FUNCTION_BLOCK DistStnArm (* Basic Function Block Type *)
  (* Standard: 61499-2 *)
  (* Version 0.2, 2003-12-04, JHC, Rockwell Automation, Renamed for better indexing. *)
  (* Compiler header: package fb.rt.wago; #include <sys/time.h> *)
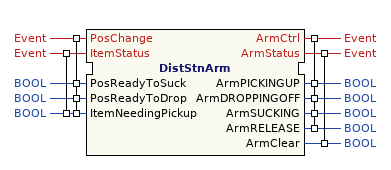
  EVENT_INPUT
    PosChange WITH PosReadyToSuck, PosReadyToDrop, ItemNeedingPickup; (* Normal Execution Request *)
    ItemStatus WITH ItemNeedingPickup;
  END_EVENT
  EVENT_OUTPUT
    ArmCtrl WITH ArmPICKINGUP, ArmDROPPINGOFF, ArmSUCKING, ArmRELEASE;
    ArmStatus WITH ArmClear; (* Execution Confirmation *)
  END_EVENT
  VAR_INPUT
    PosReadyToSuck : BOOL := false; (* Input event qualifier *)
    PosReadyToDrop : BOOL := false; (* Input event qualifier *)
    ItemNeedingPickup : BOOL;
  END_VAR
  VAR_OUTPUT
    ArmPICKINGUP : BOOL := false;
    ArmDROPPINGOFF : BOOL := false; (* Output event qualifier *)
    ArmSUCKING : BOOL := false;
    ArmRELEASE : BOOL := false;
    ArmClear : BOOL := true;
  END_VAR
  VAR
    ReleaseDelay : INT;
  END_VAR
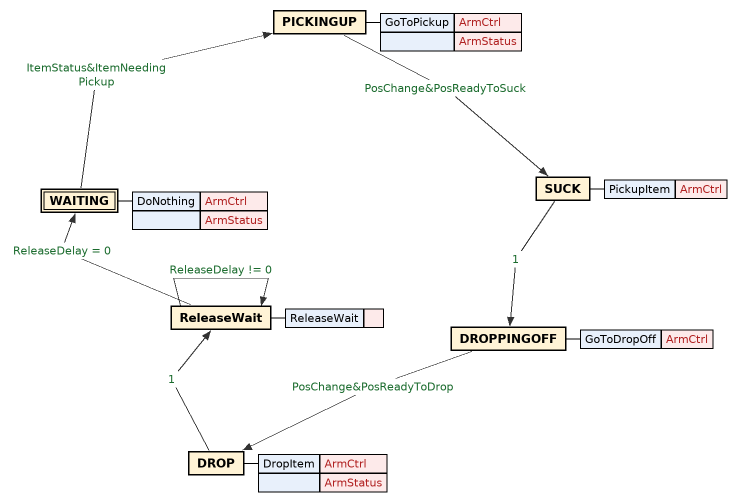
  EC_STATES
    WAITING : DoNothing -> ArmCtrl, -> ArmStatus; (* Initial State *)
    DROPPINGOFF : GoToDropOff -> ArmCtrl; (* Normal execution *)
    DROP : DropItem -> ArmCtrl, -> ArmStatus; (* Normal execution *)
    PICKINGUP : GoToPickup -> ArmCtrl, -> ArmStatus;
    SUCK : PickupItem -> ArmCtrl;
    ReleaseWait : ReleaseWait;
  END_STATES
  EC_TRANSITIONS
    WAITING TO PICKINGUP := ItemStatus&ItemNeedingPickup;
    PICKINGUP TO SUCK := PosChange&PosReadyToSuck;
    SUCK TO DROPPINGOFF := 1;
    DROPPINGOFF TO DROP := PosChange&PosReadyToDrop;
    DROP TO ReleaseWait := 1;
    ReleaseWait TO WAITING := ReleaseDelay = 0;
    ReleaseWait TO ReleaseWait := ReleaseDelay != 0;
  END_TRANSITIONS
  ALGORITHM GoToDropOff IN C: (* Initialization algorithm *)
me->ArmPICKINGUP = false;
me->ArmDROPPINGOFF = true;
  END_ALGORITHM
  ALGORITHM GoToPickup IN C: (* Initialization algorithm *)
me->ArmPICKINGUP = true;
me->ArmDROPPINGOFF = false;

me->ArmClear = false;
  END_ALGORITHM
  ALGORITHM PickupItem IN C: (* Normally executed algorithm *)
me->ArmSUCKING = true;
me->ArmRELEASE = false;
  END_ALGORITHM
  ALGORITHM CheckTimeout IN C:
//struct timeval nowtime, timediff;
//long long result;

//gettimeofday(&nowtime, NULL);
//timersub(&nowtime, &me->armTimer, &timediff);
//result = (long long)(timediff.tv_sec) * 1000000 + timediff.tv_usec;
//if( result > 1000000 )
//me->timeout = true;
  END_ALGORITHM
  ALGORITHM DropItem IN C:
me->ArmSUCKING = false;
me->ArmRELEASE = true;
me->ReleaseDelay = 5;

//gettimeofday(&me->armTimer, NULL);
//timersub(&_nowTime, &_armTimer, &timediff);


// and now we are clear

me->ArmClear = true;
  END_ALGORITHM
  ALGORITHM DoNothing IN C:
me->ArmPICKINGUP = false;
me->ArmDROPPINGOFF = false;
me->ArmSUCKING = false;
me->ArmRELEASE = false;
me->ArmClear = true;
  END_ALGORITHM
  ALGORITHM ReleaseWait IN C:
if( me->ReleaseDelay > 0 )
    (me->ReleaseDelay)--;
  END_ALGORITHM
END_FUNCTION_BLOCK
